RoboDK station: deburring.rdk

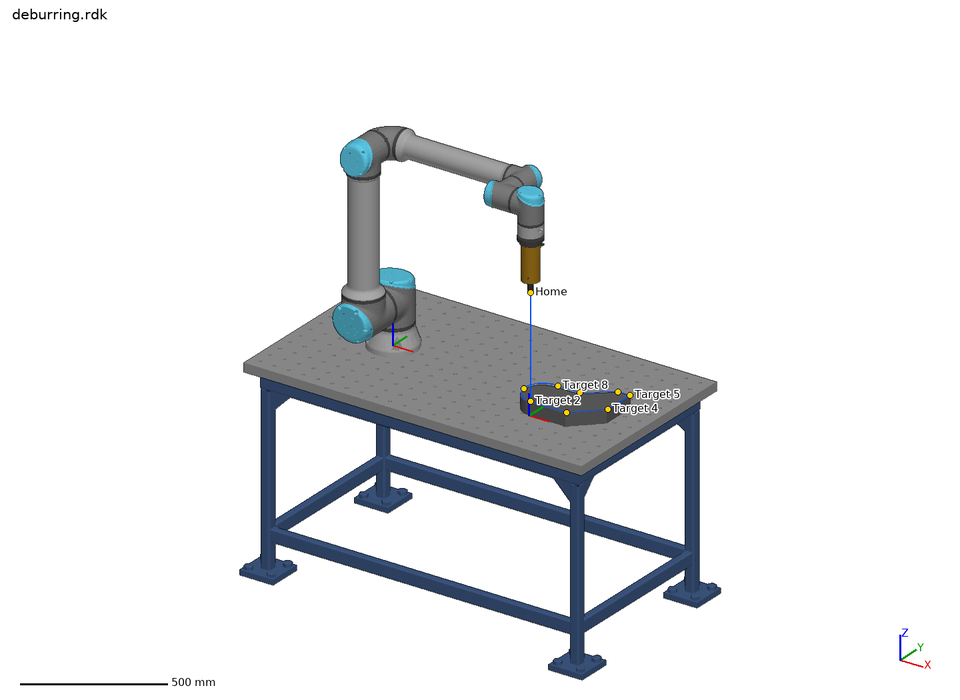
[picture v0: the station drawn from its stored meshes, robots at their saved joint values, targets as dots, program paths as lines]
Station deburring (saved by RoboDK 5.9.2). Poses are relative to the parent item; angles as X-Y-Z fixed-axis rotations.
  - frame UR10e Base at (0, 0, 0) mm
    - robot UR10e: 6 axes, payload 10 kg, reach 1300 mm, repeatability 0.05 mm, weight 28.9 kg
        modified DH rows (alpha deg, a mm, theta deg, d mm): 0, 0, 0, 180.7; 90, 0, 180, 0; 0, 612.6, 0, 0; 0, 571.335, 0, 174.15; -90, 0, 0, 119.85; 90, 0, 180, 116.55
        joint limits [-360, -360, -360, -360, -360, -360] to [360, 360, 360, 360, 360, 360]; home [0, -90, -90, 0, 90, 0]; saved at [0, -90, -90, -90, 90, 0]
      - tool ATI 9150-CDB-8-11-000 Deburring Tool (Spring), TCP at (0, 0, 215) mm, size 93.7 x 93.7 x 214.4 mm
  - object Table 1400x800x800mm at (0, 0, 0) mm, size 1420 x 820 x 800 mm, geometry from Table-1400x800x800mm.sld
  - frame Reference Frame  at (690, -180, 0) mm
    - object random1 at (0, 0, 0) mm, size 325 x 240 x 50 mm, geometry from random1.step
    - target Home (Cartesian target) at (1.19, 5.85, 461.75) mm, rotated rx -180 ry 0 rz -90 deg; joints [0, -90, -90, -90, 90, 0] of UR10e
    - target Target 2 (Cartesian target) at (1.19, 5.85, 51.75) mm, rotated rx 180 ry 0 rz -90 deg; joints [0, -104.569, -118.52, -46.911, 90, 0] of UR10e
    - target Target 3 (Cartesian target) at (151.19, 5.85, 51.75) mm, rotated rx 180 ry 0 rz -90 deg; joints [0, -115.975, -101.565, -52.461, 90, 0] of UR10e
    - target Target 4 (Cartesian target) at (251.18, 105.85, 51.75) mm, rotated rx 180 ry 0 rz -90 deg; joints [6.125, -122.627, -90.631, -56.742, 90, 6.125] of UR10e
    - target Target 5 (Cartesian target) at (251.18, 235.85, 51.75) mm, rotated rx 180 ry 0 rz -90 deg; joints [14.04, -122.527, -90.8, -56.673, 90, 14.04] of UR10e
    - target Target 6 (Cartesian target) at (201.18, 235.85, 51.75) mm, rotated rx 180 ry 0 rz -90 deg; joints [14.833, -118.604, -97.322, -54.074, 90, 14.833] of UR10e
    - target Target 7 (Cartesian target) at (101.19, 155.85, 51.75) mm, rotated rx 180 ry 0 rz -90 deg; joints [10.961, -110.761, -109.629, -49.61, 90, 10.961] of UR10e
    - target Target 8 (Cartesian target) at (11.18, 155.85, 51.75) mm, rotated rx 180 ry 0 rz -90 deg; joints [12.4, -103.669, -119.744, -46.588, 90, 12.4] of UR10e
    - target Target 9 (Cartesian target) at (-75, 75, 51.75) mm, rotated rx 180 ry 0 rz -90 deg; joints [6.52, -97.171, -128.001, -44.828, 90, 6.52] of UR10e
  - program Prog1 (12 instructions, listed below)
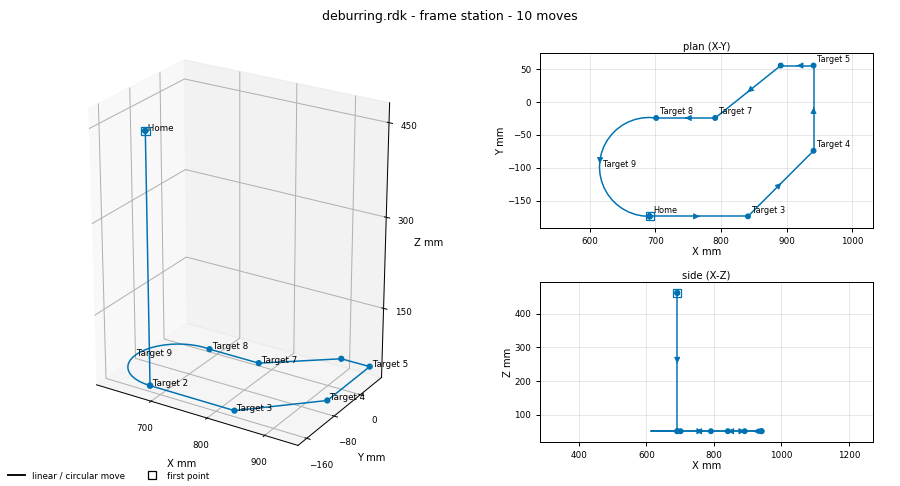
[picture p0: tool path of deburring.rdk in frame station, 10 of 10 moves have a stored position in this frame; points joined in program order, loops and branches not executed]

--- program Prog1 (robot UR10e) ---
  Set Ref.: Reference Frame -> Reference Frame 
  Set Tool: ATI 9150-CDB-8-11-000 Deburring Tool (Spring)
  MoveJ (Home)
  MoveL (Home)
  MoveL (Target 2)
  MoveL (Target 3)
  MoveL (Target 4)
  MoveL (Target 5)
  MoveL (Target 6)
  MoveL (Target 7)
  MoveL (Target 8)
  MoveC (Target 10, Target 2) -> target Target 9
